// Mitsubishi GX Works2 project: TOOL_3002_V2   PLC: FX1N/FX1NC

// global labels: Global1
VAR_GLOBAL
  Sta AT M0 : BOOL;
  Sto AT M1 : BOOL;
  Run AT M2 : BOOL;
  BX_GL AT X001 : BOOL;
  MI AT X000 : BOOL;
  BX_PK AT X002 : BOOL;
  TH AT X003 : BOOL;
  DUC1 AT X005 : BOOL;
  DUC2 AT X006 : BOOL;
  DUC3 AT X007 : BOOL;
  DUK AT X010 : BOOL;
  KA1 AT X011 : BOOL;
  KB1 AT X012 : BOOL;
  KA2 AT X013 : BOOL;
  KB2 AT X015 : BOOL;
  KAB1 AT X014 : BOOL;
  KAB2 AT X017 : BOOL;
  MI_OUT AT Y001 : BOOL;
  TH_OUT AT Y002 : BOOL;
  DUC1_OUT AT Y010 : BOOL;
  DUC3_OUT AT Y012 : BOOL;
  DUC2_OUT AT Y011 : BOOL;
  DUK_OUT AT Y013 : BOOL;
  KA1_OUT AT Y004 : BOOL;
  KB1_OUT AT Y005 : BOOL;
  KA2_OUT AT Y006 : BOOL;
  KB2_OUT AT Y007 : BOOL;
  BanXoay_ON_STATE AT M30 : BOOL;
  BanXoay_OFF_STATE AT M31 : BOOL;
  LED_ENABLE AT Y015 : BOOL;
  KB1_BUFF_1 AT M5 : BOOL;
  KA2_BUFF_1 AT M6 : BOOL;
  KB2_BUFF_1 AT M7 : BOOL;
  KB1_BUFF_13 AT M8 : BOOL;
  KB2_BUFF_13 AT M9 : BOOL;
  KA1_BUFF_1 AT M4 : BOOL;
  KA1_BUFF_2 AT M10 : BOOL;
  KB1_BUFF_2 AT M11 : BOOL;
  KA2_BUFF_2 AT M12 : BOOL;
  KB2_BUFF_2 AT M13 : BOOL;
  KB1_BUFF_23 AT M14 : BOOL;
  KB2_BUFF_23 AT M15 : BOOL;
  KA1_BUFF_12 AT M16 : BOOL;
  KA2_BUFF_12 AT M17 : BOOL;
  KB1_BUFF_12 AT M18 : BOOL;
  KB2_BUFF_12 AT M19 : BOOL;
  KA1_BUFF_22 AT M20 : BOOL;
  KB1_BUFF_22 AT M21 : BOOL;
  KA2_BUFF_22 AT M22 : BOOL;
  KB2_BUFF_22 AT M23 : BOOL;
  LENH_OUT AT Y003 : BOOL;
  ML1 AT D10 : INT;
  ML2 AT D12 : INT;
  ML3 AT D14 : INT;
  STA_RESP AT M25 : BOOL;
  ENA_BUFF AT M26 : BOOL;
END_VAR

PROGRAM MAIN
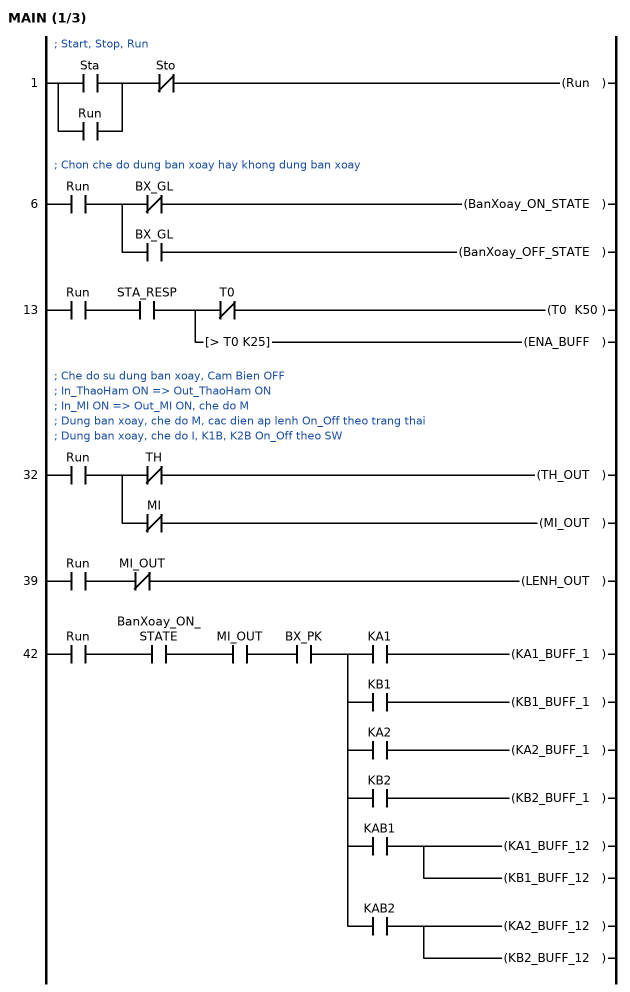
; Start, Stop, Run
1     LD      Sta
      OR      Run
      ANI     Sto
      OUT     Run
; Chon che do dung ban xoay hay khong dung ban xoay
6     LD      Run
      MPS
      ANI     BX_GL
      OUT     BanXoay_ON_STATE
      MPP
      AND     BX_GL
      OUT     BanXoay_OFF_STATE
13    LD      Run
      AND     STA_RESP
      MPS
      ANI     T0
      OUT     T0 K50
      MPP
      AND>    T0 K25
      OUT     ENA_BUFF
; Che do su dung ban xoay, Cam Bien OFF
; In_ThaoHam ON => Out_ThaoHam ON
; In_MI ON => Out_MI ON, che do M
; Dung ban xoay, che do M, cac dien ap lenh On_Off theo trang thai
; Dung ban xoay, che do I, K1B, K2B On_Off theo SW
32    LD      Run
      MPS
      ANI     TH
      OUT     TH_OUT
      MPP
      ANI     MI
      OUT     MI_OUT
39    LD      Run
      ANI     MI_OUT
      OUT     LENH_OUT
42    LD      Run
      AND     BanXoay_ON_STATE
      AND     MI_OUT
      AND     BX_PK
      MPS
      AND     KA1
      OUT     KA1_BUFF_1
      MRD
      AND     KB1
      OUT     KB1_BUFF_1
      MRD
      AND     KA2
      OUT     KA2_BUFF_1
      MRD
      AND     KB2
      OUT     KB2_BUFF_1
      MRD
      AND     KAB1
      OUT     KA1_BUFF_12
      OUT     KB1_BUFF_12
      MPP
      AND     KAB2
      OUT     KA2_BUFF_12
      OUT     KB2_BUFF_12
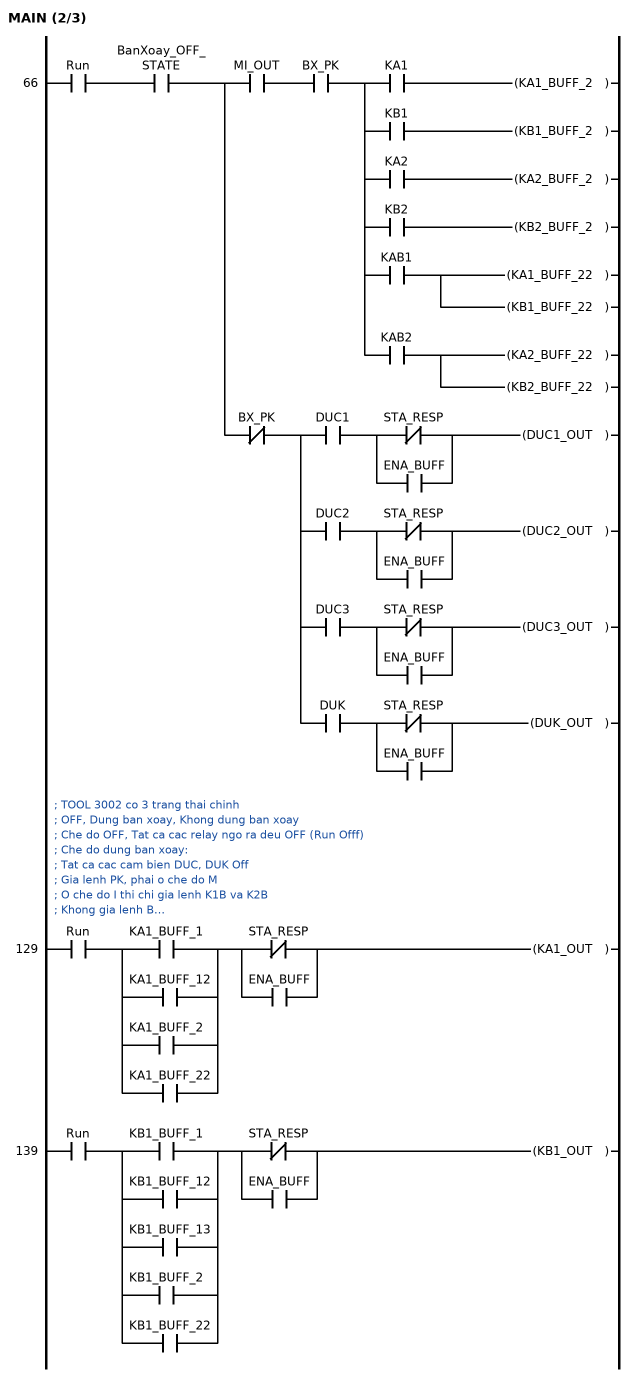
66    LD      Run
      AND     BanXoay_OFF_STATE
      MPS
      AND     MI_OUT
      AND     BX_PK
      MPS
      AND     KA1
      OUT     KA1_BUFF_2
      MRD
      AND     KB1
      OUT     KB1_BUFF_2
      MRD
      AND     KA2
      OUT     KA2_BUFF_2
      MRD
      AND     KB2
      OUT     KB2_BUFF_2
      MRD
      AND     KAB1
      OUT     KA1_BUFF_22
      OUT     KB1_BUFF_22
      MPP
      AND     KAB2
      OUT     KA2_BUFF_22
      OUT     KB2_BUFF_22
      MPP
      ANI     BX_PK
      MPS
      AND     DUC1
      LDI     STA_RESP
      OR      ENA_BUFF
      ANB
      OUT     DUC1_OUT
      MRD
      AND     DUC2
      LDI     STA_RESP
      OR      ENA_BUFF
      ANB
      OUT     DUC2_OUT
      MRD
      AND     DUC3
      LDI     STA_RESP
      OR      ENA_BUFF
      ANB
      OUT     DUC3_OUT
      MPP
      AND     DUK
      LDI     STA_RESP
      OR      ENA_BUFF
      ANB
      OUT     DUK_OUT
; TOOL 3002 co 3 trang thai chinh
; OFF, Dung ban xoay, Khong dung ban xoay
; Che do OFF, Tat ca cac relay ngo ra deu OFF (Run Offf)
; Che do dung ban xoay:
; Tat ca cac cam bien DUC, DUK Off
; Gia lenh PK, phai o che do M
; O che do I thi chi gia lenh K1B va K2B
; Khong gia lenh BX
; Che do khong dung ban xoay (Gia Bx va Pk):
; Gia lenh PK + che do M
; Gia lenh BX ca che do M va che do I
; Gia lenh Pk o che do I thi chi co K1B va K2B
129   LD      Run
      LD      KA1_BUFF_1
      OR      KA1_BUFF_12
      OR      KA1_BUFF_2
      OR      KA1_BUFF_22
      ANB
      LDI     STA_RESP
      OR      ENA_BUFF
      ANB
      OUT     KA1_OUT
139   LD      Run
      LD      KB1_BUFF_1
      OR      KB1_BUFF_12
      OR      KB1_BUFF_13
      OR      KB1_BUFF_2
      OR      KB1_BUFF_22
      ANB
      LDI     STA_RESP
      OR      ENA_BUFF
      ANB
      OUT     KB1_OUT
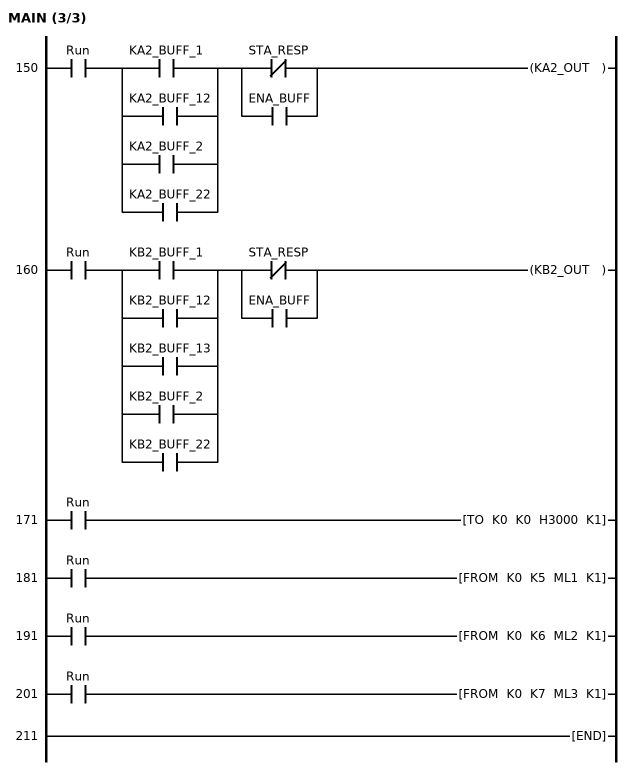
150   LD      Run
      LD      KA2_BUFF_1
      OR      KA2_BUFF_12
      OR      KA2_BUFF_2
      OR      KA2_BUFF_22
      ANB
      LDI     STA_RESP
      OR      ENA_BUFF
      ANB
      OUT     KA2_OUT
160   LD      Run
      LD      KB2_BUFF_1
      OR      KB2_BUFF_12
      OR      KB2_BUFF_13
      OR      KB2_BUFF_2
      OR      KB2_BUFF_22
      ANB
      LDI     STA_RESP
      OR      ENA_BUFF
      ANB
      OUT     KB2_OUT
171   LD      Run
      TO      K0 K0 H3000 K1
181   LD      Run
      FROM    K0 K5 ML1 K1
191   LD      Run
      FROM    K0 K6 ML2 K1
201   LD      Run
      FROM    K0 K7 ML3 K1
211   END
END_PROGRAM
